FUNCTION_BLOCK MoveMoverToPosition
VAR_INPUT
END_VAR
VAR_OUTPUT
END_VAR
VAR
	moveAbs	: MC_MoveAbsoluteCA;
	_axis : REFERENCE TO AXIS_REF;
	State: INT;
	_MoveMover : BOOL;
	_busy : BOOL;
	_error : BOOL;
	_done : BOOL;
	_stOptions : ST_MoveAbsoluteCAOptions;
END_VAR

CASE State OF
	0:
		IF _MoveMover THEN
			_done := FALSE;
			_error := FALSE;
			_busy := TRUE;
			moveAbs.Execute := TRUE;
			IF moveAbs.Busy THEN
				State := 10;
				_MoveMover := FALSE;
			END_IF
		END_IF
		
	10:
		IF NOT moveAbs.Busy THEN
			IF moveAbs.Done THEN
				_done := TRUE;
			ELSIF moveAbs.Error THEN
				_error := TRUE;
			END_IF
			_busy := FALSE;
			moveAbs.Execute := FALSE;
			State := 0;
		END_IF
END_CASE

moveAbs(Axis := _axis, Options := _stOptions);

METHOD Abort : BOOL
moveAbs.Execute := FALSE;
moveAbs.Position := moveAbs.Velocity := 0;
_MoveMover := false;
_busy := false;
Abort := true;
State := 0;
END_METHOD

PROPERTY PUBLIC Acceleration : mc_lreal
GET
Acceleration := moveAbs.Acceleration;
END_GET
SET
moveAbs.Acceleration := Acceleration;
END_SET
END_PROPERTY

PROPERTY Busy : BOOL
GET
Busy := _busy;
END_GET
END_PROPERTY

PROPERTY PUBLIC Deceleration : mc_lreal
GET
Deceleration := moveAbs.Deceleration;
END_GET
SET
moveAbs.Deceleration := Deceleration;
END_SET
END_PROPERTY

PROPERTY Done : BOOL
GET
Done := _done;
END_GET
END_PROPERTY

PROPERTY Error : BOOL
GET
Error := _error;
END_GET
END_PROPERTY

METHOD FB_init : BOOL
VAR_INPUT
	bInitRetains : BOOL; // if TRUE, the retain variables are initialized (warm start / cold start)
	bInCopyCode : BOOL;  // if TRUE, the instance afterwards gets moved into the copy code (online change)
	axis : reference TO AXIS_REF;
END_VAR
_axis REF= axis;
END_METHOD

PROPERTY PUBLIC Gap : mc_lreal
GET
Gap := moveAbs.Gap;
END_GET
SET
moveAbs.Gap := Gap;
END_SET
END_PROPERTY

PROPERTY PUBLIC Jerk : mc_lreal
GET
Jerk := moveAbs.Jerk;
END_GET
SET
moveAbs.Jerk := Jerk;
END_SET
END_PROPERTY

METHOD MoveTo : BOOL
VAR_INPUT
	Position : MC_LREAL;
	Velocity : MC_LREAL;
END_VAR
moveAbs.Position := Position;
moveAbs.Velocity := Velocity;
_MoveMover := MoveTo := true;
END_METHOD

PROPERTY PUBLIC Options : ST_MoveAbsoluteCAOptions
GET
Options := _stOptions;
END_GET
SET
_stOptions := Options;
END_SET
END_PROPERTY

END_FUNCTION_BLOCK

(* stored: Version 1.1.0.1, ProductVersion 3.1.4024.11
   POU MoveMoverToPosition: Id {7961d86e-9dbd-4bec-8af5-9f83d1007f15}, SpecialFunc None
   Method Abort: Id {f9d68d1b-cca9-4afb-b897-7620e260f1b1}
   Property Acceleration: Id {25c3f3fb-5de7-4513-80bb-e02401d941b8}
   Get Get: Id {bf7c35f7-6dac-4618-b1a4-a4c06b3b4b22}
   Set Set: Id {aa34a908-65fb-4c83-9e62-f3efb16261df}
   Property Busy: Id {6f4dca59-6db6-48ea-9403-1d24de310b7d}
   Get Get: Id {8a098c97-be03-4dd9-be2a-46f9becd37b5}
   Property Deceleration: Id {ef0b52f9-9843-49fb-a892-4640ff914923}
   Get Get: Id {bbf33e15-becc-4893-bb90-eb050f77761a}
   Set Set: Id {23b879ca-1653-4b1a-8777-f4365951865b}
   Property Done: Id {ef45dfcc-b656-4cce-b30c-b0a99f348597}
   Get Get: Id {124a0200-9a0e-40fe-b32e-4a16de2ed2e9}
   Property Error: Id {348791b2-9244-4695-bd4c-0744a35d1ffc}
   Get Get: Id {266f34a9-b654-4243-9cef-beb05b184a7d}
   Method FB_init: Id {ef6f9546-23fb-4e83-b44b-03e2dc95d5fb}
   Property Gap: Id {80e63f46-0052-47b1-bae9-3485a1a3fe8d}
   Get Get: Id {24c97301-2bd0-4413-aff6-91595a1a4944}
   Set Set: Id {f1e7e5a9-7eab-41b0-beb7-63547301c27c}
   Property Jerk: Id {fa621317-c9dd-40bb-97c3-3464fe6cb619}
   Get Get: Id {58e306a8-9f6b-4204-9666-3943ecafe1c0}
   Set Set: Id {b04b404e-8678-403b-84a1-a8e1f68db1e4}
   Method MoveTo: Id {3db5386a-5001-460e-b511-3aa21a932bfe}
   Property Options: Id {91d35b49-0fef-402f-ac14-74673db6c7d3}
   Get Get: Id {193d1496-2d7b-452f-afc5-343cbd1801df}
   Set Set: Id {51e61ca1-1574-48db-b754-cf37e5744493} *)
